// TIA Portal project "Ejercicio3-Bomba-TIA" (V14)

(* hardware
DEVICE "S7-1200 station_1"  S7-1200 Station
   slot 0: "Rack_0"  S7-1200 Rack  Rack  V1.0
   slot 1: "PLC_1"  CPU 1214C DC/DC/DC  6ES7 214-1AG40-0XB0  V4.2
*)

// ===== PLC "PLC_1"  CPU 1214C DC/DC/DC =====

VAR_GLOBAL   // PLC tag table "Tabla de variables estándar"
   "Encender" AT %I0.0 : Bool;
   "MarcaBA" AT %M0.0 : Bool;
   "MarcaBB" AT %M0.1 : Bool;
   "MarcaMA" AT %M0.2 : Bool;
   "ValvulaDeDrenaje" AT %Q0.4 : Bool;
   "Clock_Byte" AT %MB100 : Byte;
   "Clock_10Hz" AT %M100.0 : Bool;
   "Clock_5Hz" AT %M100.1 : Bool;
   "Clock_2.5Hz" AT %M100.2 : Bool;
   "Clock_2Hz" AT %M100.3 : Bool;
   "Clock_1.25Hz" AT %M100.4 : Bool;
   "Clock_1Hz" AT %M100.5 : Bool;
   "Clock_0.625Hz" AT %M100.6 : Bool;
   "Clock_0.5Hz" AT %M100.7 : Bool;
   "QBombaA" AT %Q0.0 : Bool;
   "QBombaB" AT %Q0.1 : Bool;
   "QMotorA" AT %Q0.2 : Bool;
   "QBombaC" AT %Q0.3 : Bool;
   "IndicadorBA" AT %Q0.5 : Bool;
   "IndicadorBB" AT %Q0.6 : Bool;
   "IndicadorBC" AT %Q0.7 : Bool;
   "IndicadorMA" AT %Q1.0 : Bool;
   "Error" AT %I0.1 : Bool;
   "EtiquetaError" AT %M0.3 : Bool;
   "Tag_1" AT %MD100 : Time;
END_VAR

// folder: System blocks/Program resources

DATA_BLOCK "TBOMBA1"   // DB1
{ S7_Optimized_Access := 'TRUE' }
AUTHOR : Simatic
FAMILY : IEC
NAME : IEC_TMR
VERSION : 1.0
// stored: InstanceOfName IEC_TIMER
"IEC_TIMER"
BEGIN
END_DATA_BLOCK

DATA_BLOCK "TBOMBA2"   // DB2
{ S7_Optimized_Access := 'TRUE' }
AUTHOR : Simatic
FAMILY : IEC
NAME : IEC_TMR
VERSION : 1.0
// stored: InstanceOfName IEC_TIMER
"IEC_TIMER"
BEGIN
END_DATA_BLOCK

DATA_BLOCK "TMotorAgitador"   // DB3
{ S7_Optimized_Access := 'TRUE' }
AUTHOR : Simatic
FAMILY : IEC
NAME : IEC_TMR
VERSION : 1.0
// stored: InstanceOfName IEC_TIMER
"IEC_TIMER"
BEGIN
END_DATA_BLOCK

DATA_BLOCK "TValvulaD"   // DB4
{ S7_Optimized_Access := 'TRUE' }
AUTHOR : Simatic
FAMILY : IEC
NAME : IEC_TMR
VERSION : 1.0
// stored: InstanceOfName IEC_TIMER
"IEC_TIMER"
BEGIN
END_DATA_BLOCK

DATA_BLOCK "Bomba1"   // DB5
{ S7_Optimized_Access := 'TRUE' }
AUTHOR : Simatic
FAMILY : IEC
NAME : IEC_TMR
VERSION : 1.0
// stored: InstanceOfName IEC_TIMER
"IEC_TIMER"
BEGIN
END_DATA_BLOCK

// folder: (top level)

FUNCTION "BombaA" : Void   // FC1, LAD
TITLE = Bomba A
{ S7_Optimized_Access := 'TRUE' }
VERSION : 0.1
// Salida de la Bomba y Indicador de la misma
BEGIN

REGION Network 1
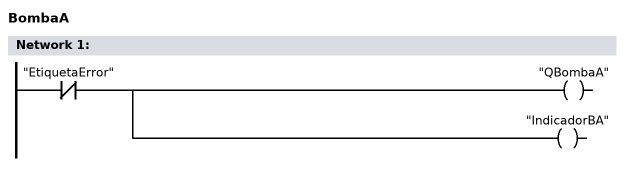
   RUNG wire#powerrail
      I_Contact( "EtiquetaError" )
      wire#w1
      Coil( "QBombaA" )
   END_RUNG
   RUNG wire#w1
      Coil( "IndicadorBA" )
   END_RUNG
   // the same network as SCL:
   "QBombaA" := NOT "EtiquetaError";
   "IndicadorBA" := NOT "EtiquetaError";
END_REGION
END_FUNCTION

FUNCTION "BombaB" : Void   // FC2, LAD
TITLE = BombaB
{ S7_Optimized_Access := 'TRUE' }
VERSION : 0.1
// Salida de la Bomba y Indicador de la misma
BEGIN

REGION Network 1
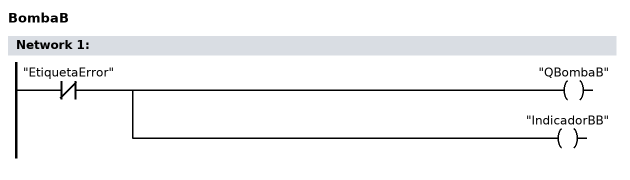
   RUNG wire#powerrail
      I_Contact( "EtiquetaError" )
      wire#w1
      Coil( "QBombaB" )
   END_RUNG
   RUNG wire#w1
      Coil( "IndicadorBB" )
   END_RUNG
   // the same network as SCL:
   "QBombaB" := NOT "EtiquetaError";
   "IndicadorBB" := NOT "EtiquetaError";
END_REGION
END_FUNCTION

FUNCTION "BombaC" : Void   // FC3, LAD
TITLE = BombaC
{ S7_Optimized_Access := 'TRUE' }
VERSION : 0.1
// Salida de la Bomba y Indicador de la misma
BEGIN

REGION Network 1
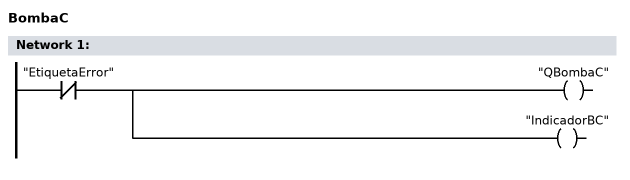
   RUNG wire#powerrail
      I_Contact( "EtiquetaError" )
      wire#w1
      Coil( "QBombaC" )
   END_RUNG
   RUNG wire#w1
      Coil( "IndicadorBC" )
   END_RUNG
   // the same network as SCL:
   "QBombaC" := NOT "EtiquetaError";
   "IndicadorBC" := NOT "EtiquetaError";
END_REGION
END_FUNCTION

FUNCTION "MotorAgitador" : Void   // FC4, LAD
{ S7_Optimized_Access := 'TRUE' }
VERSION : 0.1
BEGIN

REGION Network 1
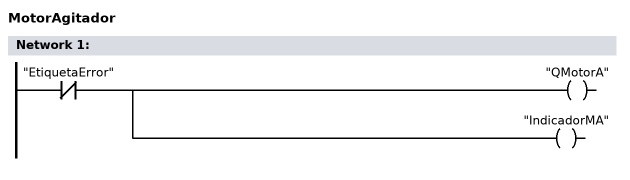
   RUNG wire#powerrail
      I_Contact( "EtiquetaError" )
      wire#w1
      Coil( "QMotorA" )
   END_RUNG
   RUNG wire#w1
      Coil( "IndicadorMA" )
   END_RUNG
   // the same network as SCL:
   "QMotorA" := NOT "EtiquetaError";
   "IndicadorMA" := NOT "EtiquetaError";
END_REGION
END_FUNCTION

FUNCTION "Alarmas" : Void   // FC5, LAD
TITLE = Alarmas
{ S7_Optimized_Access := 'TRUE' }
VERSION : 0.1
// En este bloque FC se pregunta si en el tiempo de encendido de las Bombas y el Motor, estos, se encuentran en funcionamiento. De no ser asi, se indica con el indicador de respectivo dispositivo el error a travez de un parpadeo de 1Hz, parando, ademas, todo el proceso con la etiqueta de Error.
   VAR_TEMP   // added for the SCL form of the ladder/FBD networks
      _w1 : Bool;
   END_VAR
BEGIN

REGION Network 1: AlarmaBombaA
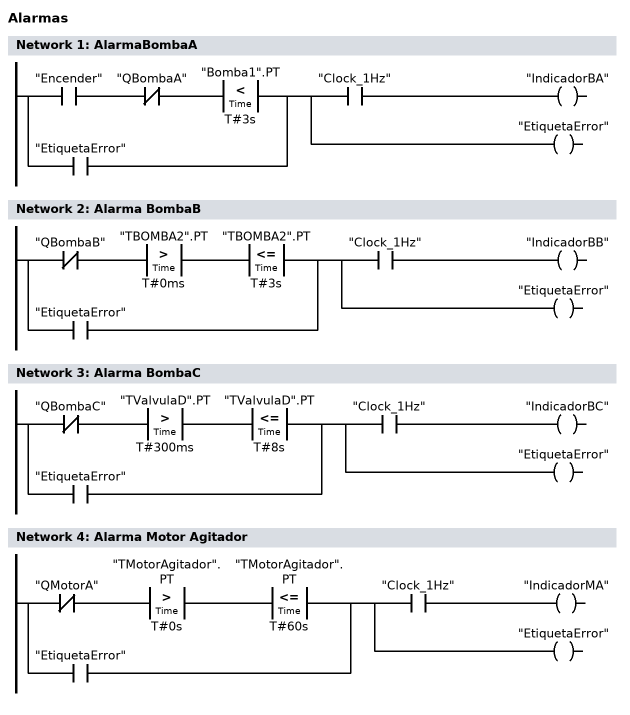
   RUNG wire#powerrail
      Contact( "Encender" )
      I_Contact( "QBombaA" )
      { S7_Templates := "SrcType := Time" } LT_Contact(in1 := "Bomba1".PT, in2 := T#3s)
      wire#w1
      Contact( "Clock_1Hz" )
      Coil( "IndicadorBA" )
   END_RUNG
   RUNG wire#powerrail
      Contact( "EtiquetaError" )
   END_RUNG wire#w1
   RUNG wire#w1
      Coil( "EtiquetaError" )
   END_RUNG
   // the same network as SCL:
   #_w1 := ("Encender" AND NOT "QBombaA" AND ("Bomba1".PT < T#3s)) OR "EtiquetaError";
   "IndicadorBA" := #_w1 AND "Clock_1Hz";
   "EtiquetaError" := #_w1;
END_REGION

REGION Network 2: Alarma BombaB
   RUNG wire#powerrail
      I_Contact( "QBombaB" )
      { S7_Templates := "SrcType := Time" } GT_Contact(in1 := "TBOMBA2".PT, in2 := T#0ms)
      { S7_Templates := "SrcType := Time" } LE_Contact(in1 := "TBOMBA2".PT, in2 := T#3s)
      wire#w1
      Contact( "Clock_1Hz" )
      Coil( "IndicadorBB" )
   END_RUNG
   RUNG wire#powerrail
      Contact( "EtiquetaError" )
   END_RUNG wire#w1
   RUNG wire#w1
      Coil( "EtiquetaError" )
   END_RUNG
   // the same network as SCL:
   #_w1 := (NOT "QBombaB" AND ("TBOMBA2".PT > T#0ms) AND ("TBOMBA2".PT <= T#3s)) OR "EtiquetaError";
   "IndicadorBB" := #_w1 AND "Clock_1Hz";
   "EtiquetaError" := #_w1;
END_REGION

REGION Network 3: Alarma BombaC
   RUNG wire#powerrail
      I_Contact( "QBombaC" )
      { S7_Templates := "SrcType := Time" } GT_Contact(in1 := "TValvulaD".PT, in2 := T#300ms)
      { S7_Templates := "SrcType := Time" } LE_Contact(in1 := "TValvulaD".PT, in2 := T#8s)
      wire#w1
      Contact( "Clock_1Hz" )
      Coil( "IndicadorBC" )
   END_RUNG
   RUNG wire#powerrail
      Contact( "EtiquetaError" )
   END_RUNG wire#w1
   RUNG wire#w1
      Coil( "EtiquetaError" )
   END_RUNG
   // the same network as SCL:
   #_w1 := (NOT "QBombaC" AND ("TValvulaD".PT > T#300ms) AND ("TValvulaD".PT <= T#8s)) OR "EtiquetaError";
   "IndicadorBC" := #_w1 AND "Clock_1Hz";
   "EtiquetaError" := #_w1;
END_REGION

REGION Network 4: Alarma Motor Agitador
   RUNG wire#powerrail
      I_Contact( "QMotorA" )
      { S7_Templates := "SrcType := Time" } GT_Contact(in1 := "TMotorAgitador".PT, in2 := T#0s)
      { S7_Templates := "SrcType := Time" } LE_Contact(in1 := "TMotorAgitador".PT, in2 := T#60s)
      wire#w1
      Contact( "Clock_1Hz" )
      Coil( "IndicadorMA" )
   END_RUNG
   RUNG wire#powerrail
      Contact( "EtiquetaError" )
   END_RUNG wire#w1
   RUNG wire#w1
      Coil( "EtiquetaError" )
   END_RUNG
   // the same network as SCL:
   #_w1 := (NOT "QMotorA" AND ("TMotorAgitador".PT > T#0s) AND ("TMotorAgitador".PT <= T#60s)) OR "EtiquetaError";
   "IndicadorMA" := #_w1 AND "Clock_1Hz";
   "EtiquetaError" := #_w1;
END_REGION
END_FUNCTION

ORGANIZATION_BLOCK "Main"   // OB1, LAD, ProgramCycle
TITLE = "Main Program Sweep (Cycle)" / Ciclo principal del Programa
{ S7_Optimized_Access := 'TRUE' }
VERSION : 0.1
// Aqui se establece la secuencia a travez de los temporizadores TP y TOF. Estos llamaran en el orden establecido a los bloques FC, en los cuales se programa la funcion de encender el motor y bombas eh indicar, a travez de un Led Indicador, su estado On/Off. 
//       Se llama en el Segmento 2, el bloque de funcion FC5 Alarmas.
   VAR_INPUT
      Initial_Call : Bool;   // Initial call of this OB
      Remanence : Bool;   // =True, if remanent data are available
   END_VAR
BEGIN

REGION Network 1: Secuencia
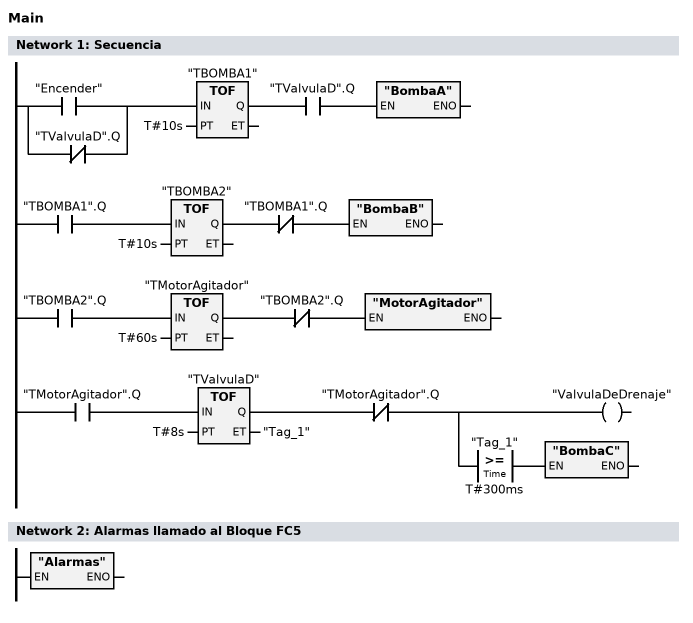
   "TBOMBA1".TOF(IN := "Encender" OR NOT "TValvulaD".Q, PT := T#10s);
   IF "TBOMBA1".Q AND "TValvulaD".Q THEN "BombaA"(); END_IF;
   "TBOMBA2".TOF(IN := "TBOMBA1".Q, PT := T#10s);
   IF "TBOMBA2".Q AND NOT "TBOMBA1".Q THEN "BombaB"(); END_IF;
   "TMotorAgitador".TOF(IN := "TBOMBA2".Q, PT := T#60s);
   IF "TMotorAgitador".Q AND NOT "TBOMBA2".Q THEN "MotorAgitador"(); END_IF;
   "TValvulaD".TOF(IN := "TMotorAgitador".Q, PT := T#8s, ET => "Tag_1");
   "ValvulaDeDrenaje" := "TValvulaD".Q AND NOT "TMotorAgitador".Q;
   IF "ValvulaDeDrenaje" AND ("Tag_1" >= T#300ms) THEN "BombaC"(); END_IF;
END_REGION

REGION Network 2: Alarmas llamado al Bloque FC5
   RUNG wire#powerrail
      "Alarmas"()
   END_RUNG
   // the same network as SCL:
   "Alarmas"();
END_REGION
END_ORGANIZATION_BLOCK